Staubli VAL3: bmask.pgx

public program bmask(num x_mask, num& x_return[])
// Create binary mask
begin
  x_return=exp(roundDown(x_mask)*ln(2))
  if bDebug
    putln("bmask(): "+toString("0.0",x_mask)+" => "+toString("0.0",x_return))
  endIf
end
